// TIA Portal V17 export
// export: Created 2024-10-17T14:16:17.167416Z, ExportSetting WithDefaults, DisplayName Totally Integrated Automation Portal, DisplayVersion V17 Update 4, DisplayName TIA Portal Openness, DisplayVersion V17 Update 4, DisplayName TIA Portal Version Control Interface, DisplayVersion V17, DisplayName SINAMICS Startdrive Advanced, DisplayVersion V17 Update2, DisplayName SINAMICS Startdrive G130, G150, S120, S150, SINAMICS MV, S210, DisplayVersion V17 Update2, DisplayName SINAMICS Startdrive G110M, G120, G120C, G120D, G120P, G115D, DisplayVersion V17 Update2, DisplayName STEP 7 Professional, DisplayVersion V17 Update 4, DisplayName STEP 7 Safety, DisplayVersion V17, DisplayName WinCC Advanced / Unified PC, DisplayVersion V17 Update 4
TYPE "LPMLV2022_typeStatus"
TITLE = LPMLV2022_typeStatus
// Support: tech.team.motioncontrol@siemens.com
// stored: IsFailsafeCompliant false
   STRUCT
      UnitModeCurrent { ExternalWritable := 'False'} : DInt;   // Current Unit Mode Number (0: Invalid, 1: Production, 2: Maintenance, 3: Manual, 04 - 31: User Definable). Minimum required for information/machine monitoring
      UnitModeRequested { ExternalWritable := 'False'} : Bool;   // Requested Unit Mode Change. When a unit mode request takes place a numerical value must be present in the unit mode target to change the unit mode
      UnitModeChangeInProcess { ExternalWritable := 'False'} : Bool;   // Requested Unit Mode Change In Process
      StateCurrent { ExternalWritable := 'False'} : DInt;   // Current State Number (0: Undefined, 1: CLEARING, 2: STOPPED, 3: STARTING, 4: IDLE, 5: SUSPENDED, 6: EXECUTE, 7: STOPPING, 8: ABORTING, 9: ABORTED; 10: HOLDING, 11: HELD, 12: UNHOLDING, 13: SUSPENDING, 14: UNSUSPENDING, 15: RESETTING, 16: COMPLETING, 17: COMPLETED). Minimum required for information/machine monitoring
      StateRequested { ExternalWritable := 'False'} : DInt;   // Target State. This value is used for state transition checking, to ensure that transition to a target state can be achieved
      StateChangeInProcess { ExternalWritable := 'False'} : Bool;   // State Change in Process. This bit indicates that a change in state is in progress following a state change request command
      MachSpeed { ExternalWritable := 'False'} : Real;   // Current Machine Speed Setpoint. This describes the set point for the current speed of the machine in primary packages per minute. Minimum required for information/machine monitoring
      CurMachSpeed { ExternalWritable := 'False'} : Real;   // Current Actual Machine Speed. This is the actual value of the machine speed in primary packages per minute. Minimum required for information/machine monitoring
      MaterialInterlock { ExternalWritable := 'False'} : DWord;   // Materials Ready. MaterialInterlock describes the status of the materials that are ready for processing. It is comprised of a series of bits with 1 equaling ready or not low, 0 equaling not ready, or low. Each bit represents a different user material
      EquipmentInterlock { ExternalWritable := 'False'} : "LPMLV2022_typeEquipmentInterlock";   // Is a collection of tags that are used to provide an indicator of Blocked or Starved conditions at the machine unit when integrated into a complete production line
      Parameter_REAL { ExternalWritable := 'False'} : Array[0.."LPMLV2022_STATUS_PARAMETER_REAL_UPPER_LIM"] of "LPMLV2022_typeParameter_REAL";   // Structured Array of Unit/Machine Parameter information for values with REAL data type
      Parameter_STRING { ExternalWritable := 'False'} : Array[0.."LPMLV2022_STATUS_PARAMETER_STRING_UPPER_LIM"] of "LPMLV2022_typeParameter_STRING";   // Structured Array of Unit/Machine Parameter information for values with STRING data type
      Parameter_LREAL { ExternalWritable := 'False'} : Array[0.."LPMLV2022_STATUS_PARAMETER_LREAL_UPPER_LIM"] of "LPMLV2022_typeParameter_LREAL";   // Structured Array of Unit/Machine Parameter information for values with LREAL data type
      Parameter_DINT { ExternalWritable := 'False'} : Array[0.."LPMLV2022_STATUS_PARAMETER_DINT_UPPER_LIM"] of "LPMLV2022_typeParameter_DINT";   // Structured Array of Unit/Machine Parameter information for values with DINT data type
      Parameter_BOOL { ExternalWritable := 'False'} : Array[0.."LPMLV2022_STATUS_PARAMETER_BOOL_UPPER_LIM"] of "LPMLV2022_typeParameter_BOOL";   // Structured Array of Unit/Machine Parameter information for values with BOOL data type
      RecipeCurrent { ExternalWritable := 'False'} : DInt;   // The recipe currently running in production
      RecipeRequested { ExternalWritable := 'False'} : DInt;   // A reflection of the recipe currently selected for production
      RecipeChangeInProcess { ExternalWritable := 'False'} : Bool;   // An indicator for the user-defined recipe changeover process
      Recipe { ExternalWritable := 'False'} : Array[0.."LPMLV2022_STATUS_RECIPE_UPPER_LIM"] of "LPMLV2022_typeStatusRecipe";   // Structured Array of Recipe Information. The recipe data type can be used for defining product ingredient and product processing parameter variables
      Stacklight { ExternalWritable := 'False'} : Array[0.."LPMLV2022_STATUS_STACK_LIGHT_UPPER_LIM"] of DWord;   // Indicator for the current stacklight status. This tag can be used simultaneously for reporting stacklight conditions and as control bits for physical outputs. The status of a light in the stack is associated to a particular bit location within the register (Bit 0: Red Solid, 1: Red Flashing, 2: Amber Solid, 3: Amber Flashing, 4: Blue Solid, 5: Blue Flashing, 6: Green Solid, 7: Green Flashing, 8: Horn Solid, 9: Horn Flashing, 10..31: User-Defined)
   END_STRUCT;
END_TYPE
